FUNCTION_BLOCK PUBLIC MOtionControlEXT EXTENDS MotionControl
VAR_INPUT
END_VAR
VAR_OUTPUT
END_VAR
VAR
END_VAR

END_FUNCTION_BLOCK

(* stored: Version 1.1.0.1, ProductVersion 3.1.0.36
   POU MOtionControlEXT: Id {2cd156df-35e5-41ef-8fc5-c19aca351a71}, SpecialFunc None *)
